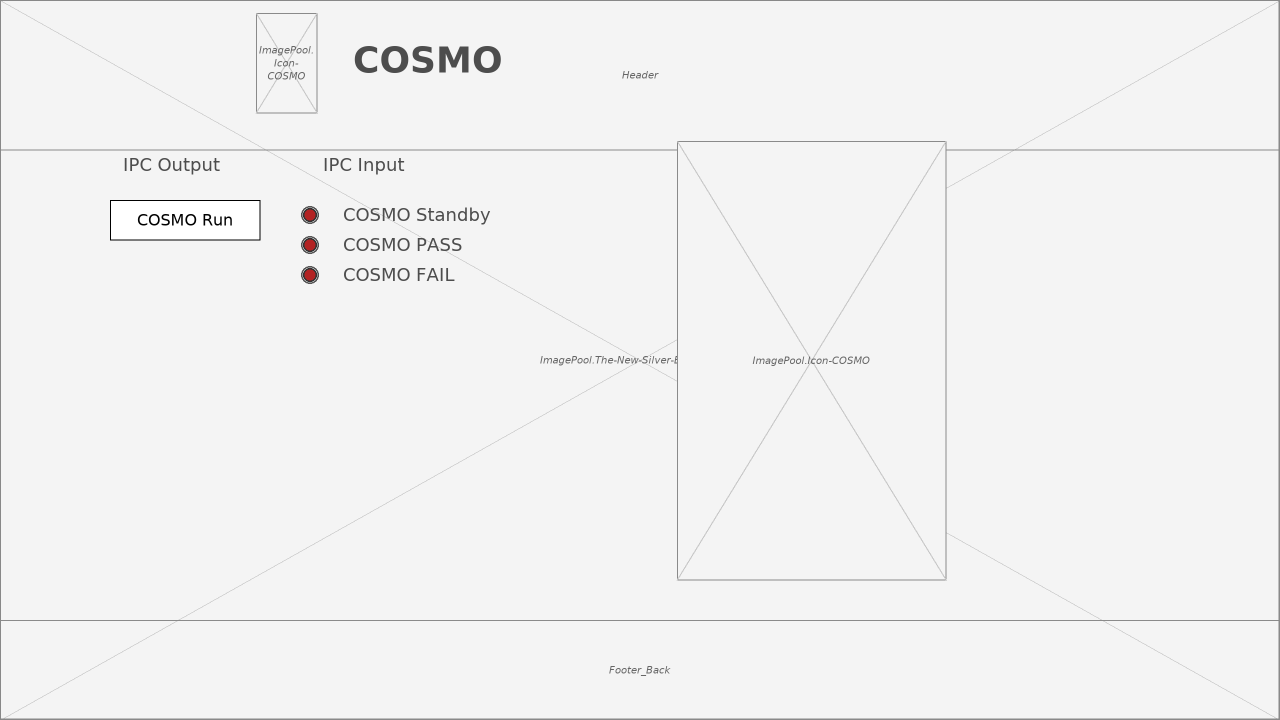
VISUALIZATION PAGE_COSMO  // 1280x720
    Image (0,0 1280x720), image: ImagePool.The-New-Silver-Backgrounds
    Frame (0,620 1280x100)
        shows Footer_Back()
    Frame (0,0 1280x150)
        shows Header()
    Label (350,40 300x40), "COSMO"
    Label (120,150 150x30), "IPC Output"
    Label (320,150 150x30), "IPC Input"
    Label (340,200 170x30), "COSMO Standby"
    Lamp1 (300,205 20x20), variable: GVL.COSMO_Ready, style: Lamp-Lamp1-Red
    Label (340,230 170x30), "COSMO PASS"
    Lamp1 (300,235 20x20), variable: GVL.COSMO_OK, style: Lamp-Lamp1-Red
    Label (340,260 170x30), "COSMO FAIL"
    Lamp1 (300,265 20x20), variable: GVL.COSMO_NOTOK, style: Lamp-Lamp1-Red
    RoundedRectangle (110,200 150x40), "COSMO Run"
        toggle GVL.COSMO_Run
    Image (256,13 61x100), image: ImagePool.Icon-COSMO
    Image (677,141 269x439), image: ImagePool.Icon-COSMO
END_VISUALIZATION

(* stored: Version 1.1.0.1, ProductVersion 3.1.4024.12
   Visu PAGE_COSMO: Id {4c08e5d4-3c7d-4452-a42a-77adce237e5a} *)
